{attribute addProperty BoxType "ATH2000-0250-0023"}
{attribute addProperty Id "A_0015_ATH2040_5250_0022ATH2040_D9917BEB11214"}
{attribute addProperty CRC "6493397"}
{attribute addProperty SizeInBites "112"}
{attribute addProperty SizeInBytes "14"}
TYPE A_0002_ATH2000_0250_0023_006314D5 EXTENDS ATH2000_9506A482 :
STRUCT
	{attribute addProperty Name "A_0015_ATH2040_5250_0022"}
	A_0015_ATH2040_5250_0022 : ATH2040_D9917BEB;
END_STRUCT
END_TYPE

(* stored: Version 1.2.0.0, ProductVersion 3.1.4024.9
   DUT A_0002_ATH2000_0250_0023_006314D5: Id {b38235ba-fcd0-41f4-a054-ba80e782be34} *)
